FUNCTION_BLOCK MAX_FB
VAR_INPUT
	In1: LREAL;
	In2: LREAL;
END_VAR
VAR_OUTPUT
	Out: LREAL;
END_VAR
VAR
END_VAR

Out := MAX(In1, In2);

END_FUNCTION_BLOCK

(* stored: Version 1.1.0.1, ProductVersion 3.1.4024.3
   POU MAX_FB: Id {d82ba786-bb4e-46e1-9dfd-243071a344a6}, SpecialFunc None *)
